INTERFACE I_PersistentEventStorage

METHOD StoreEvent
VAR_INPUT
	stEvent : ST_Event;
END_VAR
END_METHOD

END_INTERFACE

(* stored: Version 1.1.0.1, ProductVersion 3.1.4024.12
   Itf I_PersistentEventStorage: Id {018befa4-1635-4e34-ae5c-abc0433789c4}
   Method StoreEvent: Id {b5a8a6f9-0819-4ef1-8d47-46add9089518} *)
